// Mitsubishi GX Developer project: B-3-1   PLC: FX2N

PROGRAM Main
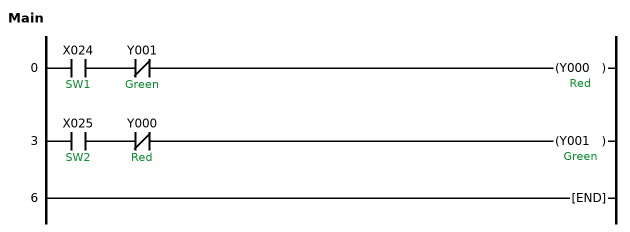
0     LD      X024  ; SW1
      ANI     Y001  ; Green
      OUT     Y000  ; Red
3     LD      X025  ; SW2
      ANI     Y000  ; Red
      OUT     Y001  ; Green
6     END
END_PROGRAM
